(* PLC project motor_project.project, CODESYS CODESYS V3.5 SP8 Patch 2 *)
(* stored: creationDateTime 2016-04-24T17:57:33.415311, modificationDateTime 2016-04-24T17:42:05.1952198 *)

PROGRAM Motion_ST
  VAR
    state : INT := 1;
    Distance : LREAL := 360;
    PowerX : MC_Power;
    Xonb : BOOL;
    HomeX : MC_Home;
    Referenced : BOOL;
    ExtendX : MC_MoveRelative;
    Wait : TON;
    RetractX : MC_MoveAbsolute;
    Wait_time : TIME := TIME#3s0ms;
    Elapsed_time : TIME;
    ResetX : MC_Reset;
    ReadAxisState : MC_ReadStatus;
    Xerrorstop : BOOL;
    XerrorID : DWORD;
    Counter : INT := 0;
  END_VAR
  VAR CONSTANT
    ERROR : INT := 99;
  END_VAR

                    
CASE state OF
	
1:
PowerX(
	Axis:=MyMotor , 
	Enable:=TRUE , 
	bRegulatorOn:=TRUE , 
	bDriveStart:=TRUE , 
	Status=> , 
	bRegulatorRealState=> , 
	bDriveStartRealState=> , 
	Busy=> , 
	Error=> , 
	ErrorID=> );
	
	IF PowerX.bDriveStartRealState THEN
		Xonb:=TRUE;
		state:=state+1;
		ELSE
			state:=ERROR;
	END_IF
	
2:
HomeX(
	Axis:=MyMotor , 
	Execute:=TRUE, 
	Position:=0.0, 
	Done=> , 
	Busy=> , 
	CommandAborted=> , 
	Error=> , 
	ErrorID=> );
		
	IF HomeX.Done THEN
		Referenced:=TRUE;
		state:=state+1;
		HomeX.Execute:=FALSE;
		ELSIF HomeX.Error OR Xerrorstop OR MyMotor.bError THEN
		state:=ERROR;
	END_IF
	
3:
ExtendX.Execute:=TRUE; 
ExtendX.Distance:=Distance; 
ExtendX.Velocity:=100; 
ExtendX.Acceleration:=1000; 
ExtendX.Deceleration:=1000; 
ExtendX.Jerk:=0; 

	IF ExtendX.Done THEN
		state:=state+1;
		ExtendX.Execute:=FALSE;
		ELSIF ExtendX.Error OR Xerrorstop OR MyMotor.bError THEN
		state:=ERROR;	
	END_IF
	
4:
Wait.IN:=TRUE;
Wait.PT:=Wait_time;
Elapsed_time:=Wait.ET;

	IF Wait.Q THEN
		state:=state+1;
		Wait.IN:=FALSE;
	END_IF

5: 
RetractX.Execute:=TRUE; 
RetractX.Position:=0; 
RetractX.Velocity:=100;
RetractX.Acceleration:=1000;
RetractX.Deceleration:=1000; 
RetractX.Jerk:=0; 

IF RetractX.Done THEN
		state:=state+1;
		RetractX.Execute:=FALSE;
		counter:=counter+1;
		ELSIF RetractX.Error OR Xerrorstop THEN
		state:=ERROR;
	END_IF
	
6: 
Wait.IN:=TRUE; 
Wait.PT:=Wait_time;
Elapsed_time:=Wait.ET;

	IF Wait.Q THEN
		state:=3;
		Wait.IN:=FALSE;
	END_IF
	
ERROR:
ResetX.Execute:=TRUE;
Wait.IN:=TRUE;
IF Wait.Q THEN
	ResetX.Execute:=FALSE;
	state:=1;
END_IF

END_CASE
ExtendX(Axis:=MyMotor);
Wait();
RetractX(Axis:=MyMotor);
ResetX(Axis:=MyMotor);
ReadAxisState(Axis:=MyMotor,Enable:=TRUE,ErrorStop=>Xerrorstop);




                  
END_PROGRAM

PROGRAM Motor_Proba
  VAR_INPUT
    START AT %MX0.1 : BOOL := FALSE;
    STOP AT %MX0.2 : BOOL := FALSE;
  END_VAR
  VAR
    MOTOR AT %MX1.0 : BOOL := FALSE;
    ERROR AT %MX2.0 : BOOL := FALSE;
  END_VAR
  VAR
    ERR_TIM : TON;
    EL_TIME : TIME;
  END_VAR
  VAR_OUTPUT
    ST_RED AT %QX1.1 : BOOL;
    ST_GREEN AT %QX3.1 : BOOL;
  END_VAR

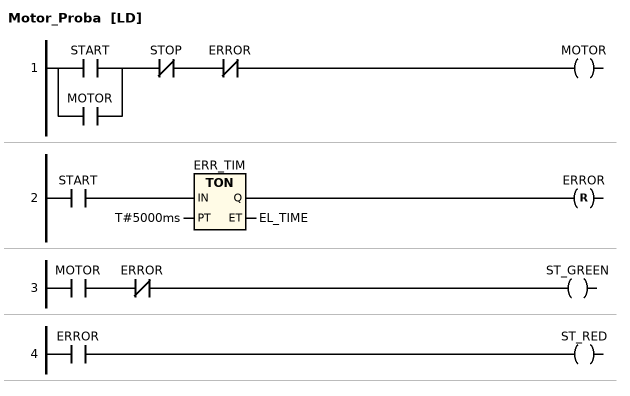
(* LD diagram, written out as Structured Text *)

MOTOR := (START OR MOTOR) AND NOT STOP AND NOT ERROR;

ERR_TIM(IN := START, PT := T#5000ms, ET => EL_TIME);
IF ERR_TIM.Q THEN ERROR := FALSE; END_IF;

ST_GREEN := MOTOR AND NOT ERROR;

ST_RED := ERROR;
END_PROGRAM

CONFIGURATION Only_motor_only_simulation
  RESOURCE Application ON PLC
    TASK ExampleTask(INTERVAL := T#10ms, PRIORITY := 1);
    PROGRAM Motor_Proba WITH ExampleTask : Motor_Proba;
    PROGRAM Motion_ST WITH ExampleTask : Motion_ST;
  END_RESOURCE
END_CONFIGURATION
